// TIA Portal V20 export
FUNCTION_BLOCK "AutoIndication"   // FB300, FBD
{ S7_Optimized_Access := 'TRUE' }
// stored: AutoNumber false, MemoryReserve 100, SetENOAutomatically false
   VAR DB_SPECIFIC
      Var { ExternalAccessible := 'False'; ExternalVisible := 'False'; ExternalWritable := 'False'} : "TypeVar";
      T { ExternalAccessible := 'False'; ExternalVisible := 'False'; ExternalWritable := 'False'} : Array[1..5] of IEC_TIMER;
   END_VAR
BEGIN

REGION Network 1: lamp test
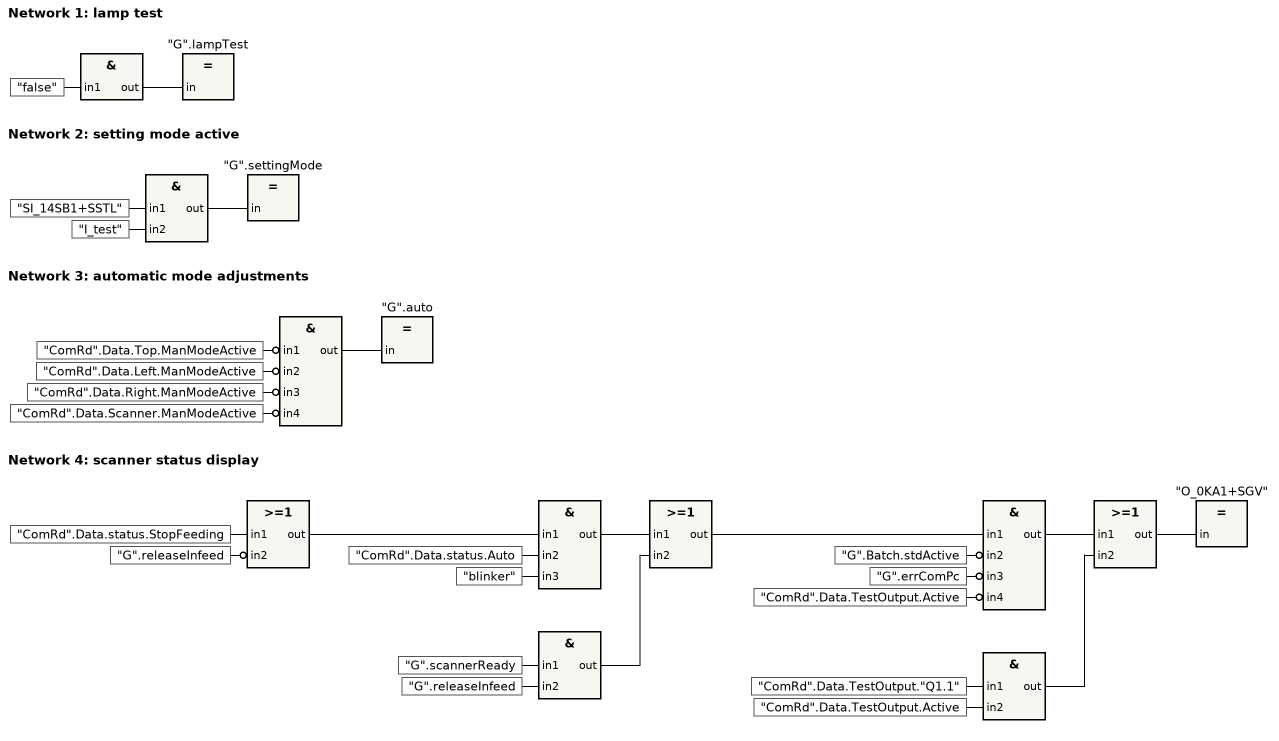
   "G".lampTest := "false";
END_REGION

REGION Network 2: setting mode active
   "G".settingMode := "SI_14SB1+SSTL" AND "I_test";
END_REGION

REGION Network 3: automatic mode adjustments
   "G".auto := NOT "ComRd".Data.Top.ManModeActive AND NOT "ComRd".Data.Left.ManModeActive AND NOT "ComRd".Data.Right.ManModeActive AND NOT "ComRd".Data.Scanner.ManModeActive;
END_REGION

REGION Network 4: scanner status display
   "O_0KA1+SGV" := (((("ComRd".Data.status.StopFeeding OR NOT "G".releaseInfeed) AND "ComRd".Data.status.Auto AND "blinker") OR ("G".scannerReady AND "G".releaseInfeed)) AND NOT "G".Batch.stdActive AND NOT "G".errComPc AND NOT "ComRd".Data.TestOutput.Active) OR ("ComRd".Data.TestOutput."Q1.1" AND "ComRd".Data.TestOutput.Active);
END_REGION
END_FUNCTION_BLOCK
